PROGRAM MAIN
VAR
END_VAR

END_PROGRAM

(* stored: Version 1.1.0.1
   POU MAIN: Id {b4091923-fc6d-4f6e-92cc-aaaf103c544c} *)
